// TwinCAT 3 PLC project PRG_B_Base_HMI
// Title: B_Base_HMI_Connector
// Company: RafalOS
// Author: Rafał Osajda
// ProjectVersion: 0.0.0.16
// ProgramVersion: 3.1.4026.18
// libraries:
//   B_Base, * (RafalOS)
//   Tc2_Standard, * (Beckhoff Automation GmbH)
//   Tc2_System, * (Beckhoff Automation GmbH)
//   Tc3_Module, * (Beckhoff Automation GmbH)
// project tree:
//   / PlcTask.TcTTO
//   POUs Compilation/ PRG_Compilation.TcPOU
//   POUs/A02_FB_BaseLogger_HMI/ FB_BaseLogger_HMI.TcPOU, ITF_BaseLogger_HMI.TcIO, ST_BaseLogger_HMI.TcDUT
//   POUs/A03_FB_BaseLoggerElement_HMI/ FB_BaseLoggerElement_HMI.TcPOU, ITF_BaseLoggerElement_HMI.TcIO, ST_BaseHMIConnectorEvents_ActionButtuns.TcDUT, ST_BaseHMIConnectorEvents_DetailInformation.TcDUT (not stored), ST_BaseHMIConnectorEvents_Filter.TcDUT, ST_BaseHMIConnectorEvents_ListToDisplay.TcDUT, ST_BaseLoggerElement_HMI.TcDUT, ST_BaseHMIConnectorEvents_ListToDisplayRow.TcDUT
//   POUs/A04_FB_BaseComponent_HMI/ FB_BaseComponent_HMI.TcPOU, ITF_BaseComponent_HMI.TcIO, ST_BaseComponent_HMI.TcDUT, ST_BaseComponent_HMI_Link.TcDUT
//   POUs/A05_FB_BaseControlElement_HMI/ FB_BaseControlElement_HMI.TcPOU, ITF_BaseControlElement_HMI.TcIO, ST_BaseControlElement_HMI.TcDUT, ST_BaseControlElement_HMI_Link.TcDUT
//   POUs/A06_FB_BaseGroupElement_HMI/ FB_BaseGroupElement_HMI.TcPOU, ITF_BaseGroupElement_HMI.TcIO, ST_BaseGroupElement_HMI.TcDUT, ST_BaseGroupElement_HMI_Link.TcDUT
//   POUs/A07_FB_BaseTopElement_HMI/ FB_BaseTopElement_HMI.TcPOU, ITF_BaseTopElement_HMI.TcIO, ST_BaseTopElement_HMI.TcDUT, ST_BaseTopElement_HMI_Link.TcDUT (not stored)

CONFIGURATION PRG_B_Base_HMI
    RESOURCE PLC ON TwinCAT3
        TASK PlcTask(INTERVAL := T#10ms, PRIORITY := 20);
        PROGRAM PRG_Compilation WITH PlcTask : PRG_Compilation;
    END_RESOURCE
END_CONFIGURATION

// ---- POUs/A02_FB_BaseLogger_HMI/ST_BaseLogger_HMI.TcDUT
TYPE ST_BaseLogger_HMI :
STRUCT
	bDanaBaseLogger		: BOOL;
END_STRUCT
END_TYPE

// ---- POUs/A03_FB_BaseLoggerElement_HMI/ST_BaseHMIConnectorEvents_ActionButtuns.TcDUT
(*			
	EVERDE sp. z o.o.
	Rafał Osajda		07.10.2025		TC 4024.66
	Przyciski akcji w zgłoszeniach zatwierdzanie zamykanie
*)
TYPE ST_BaseHMIConnectorEvents_ActionButtuns :
STRUCT
	bAcknowledgeAll				: BOOL;
	bAcknowledgeAllActive		: BOOL;		//widoczność przycisku 
	sAcknowledgeAll				: STRING;	//ilosci 

	bCloseAll					: BOOL;
	bCloseAllActive				: BOOL;		//widoczność przycisku 
	sCloseAll					: STRING;	//ilosci 
	
	bAcknowledgeSelected		: BOOL;
	bAcknowledgeSelectedActive	: BOOL;		//widoczność przycisku 
	sAcknowledgeSelected		: STRING;

	bCloseSelected				: BOOL;
	bCloseSelectedActive		: BOOL;		//widoczność przycisku 
	sCloseSelected				: STRING;	//ilosci 
END_STRUCT
END_TYPE

// ---- POUs/A03_FB_BaseLoggerElement_HMI/ST_BaseHMIConnectorEvents_Filter.TcDUT
TYPE ST_BaseHMIConnectorEvents_Filter :
STRUCT
	bActive						: BOOL;
	bNotActive					: BOOL;
	
	bIDItem						: BOOL;
	uiIDItem					: UINT;
	
	bIDEvent					: BOOL;
	uiIDEvent					: UINT;
	
	arrSelectedEventCategory	: ARRAY [0..GVL_BaseConstans.NUMBER_OF_EVENT_CATEGORIES] OF BOOL;	//przyciski selektora kategorii zdarzen - czy nacisniety
	arrTextOnEventCategory		: ARRAY [0..GVL_BaseConstans.NUMBER_OF_EVENT_CATEGORIES] OF STRING;	//teksty na przyciskach 
	
END_STRUCT
END_TYPE

// ---- POUs/A03_FB_BaseLoggerElement_HMI/ST_BaseHMIConnectorEvents_ListToDisplay.TcDUT
TYPE ST_BaseHMIConnectorEvents_ListToDisplay :
STRUCT
	arrToDisplay				: ARRAY [1..GVL_BaseConstans.MAX_EVENTS_TO_SHOW] OF ST_BaseHMIConnectorEvents_ListToDisplayRow;
	iNumberOfRow				: INT;
	bSelected					: BOOL;

END_STRUCT
END_TYPE

// ---- POUs/A03_FB_BaseLoggerElement_HMI/ST_BaseLoggerElement_HMI.TcDUT
TYPE ST_BaseLoggerElement_HMI :
STRUCT
	stFilter						: ST_BaseHMIConnectorEvents_Filter;
	stListOfEventsToDisplay			: ST_BaseHMIConnectorEvents_ListToDisplay;
	stButtons						: ST_BaseHMIConnectorEvents_ActionButtuns;
	stDetailInformation				: ST_BaseHMIConnectorEvents_DetailInformation;
	bSelected						: BOOL;
	iSelectedRow					: INT;
	iSelectedRowPrevius				: INT;
	bRefreshInfo					: BOOL;
	bRefreshList					: BOOL;
	
END_STRUCT
END_TYPE

// ---- POUs/A03_FB_BaseLoggerElement_HMI/ST_BaseHMIConnectorEvents_ListToDisplayRow.TcDUT
TYPE ST_BaseHMIConnectorEvents_ListToDisplayRow :
STRUCT
	uiIDEvent						: UINT;
	uiIDItem						: UINT;				//id elementu
	sCode							: STRING;			//kod elementu
	bActive							: BOOL;
	bIgnoreRepetitions				: BOOL;				//jak true nie zliczaj powtorzeń wystapienia np komunikaty
	uiRepetitionCounter				: UINT;
	sStart							: STRING;			//poczatek wystepowania zgłoszenia
	sFinish							: STRING;			//koniec wystepowaniazgloszenia
	sConfirmed						: STRING;			// stempel potwierdzenia 
	bConfirm						: BOOL;				//informacja czy potrzebne jest potwierdzenie 
	bConfirmed						: BOOL;				//pamięta czy już potwierdzone
	sEventCategory					: STRING;
	wsDescription					: WSTRING;
	wsDescriptionFull				: WSTRING;
	wsNameOfitem					: WSTRING;
END_STRUCT
END_TYPE

// ---- POUs/A04_FB_BaseComponent_HMI/ST_BaseComponent_HMI.TcDUT
TYPE ST_BaseComponent_HMI :
STRUCT
	bDanaBaseComponent		: BOOL;
	
END_STRUCT
END_TYPE

// ---- POUs/A04_FB_BaseComponent_HMI/ST_BaseComponent_HMI_Link.TcDUT
(*			
	RAFALOS
	Rafał Osajda		23.09.2025		TC 4024.66
	Struktura pomocnicza potrzeba do wiazania zmiennych
*)
TYPE ST_BaseComponent_HMI_Link :
STRUCT
	stBaseLoggerElement				: ST_BaseLoggerElement_HMI;
	stBaseComponent					: ST_BaseComponent_HMI;
END_STRUCT
END_TYPE

// ---- POUs/A05_FB_BaseControlElement_HMI/ST_BaseControlElement_HMI.TcDUT
TYPE ST_BaseControlElement_HMI :
STRUCT
	bDanaBaseControlElement		: BOOL;
	
END_STRUCT
END_TYPE

// ---- POUs/A05_FB_BaseControlElement_HMI/ST_BaseControlElement_HMI_Link.TcDUT
(*			
	RAFALOS
	Rafał Osajda		23.09.2025		TC 4024.66
	Struktura pomocnicza potrzeba do wiazania zmiennych
*)
TYPE ST_BaseControlElement_HMI_Link :
STRUCT
	stBaseLoggerElement				: ST_BaseLoggerElement_HMI;
	stBaseComponent					: ST_BaseComponent_HMI;
	stBaseControlElement			: ST_BaseControlElement_HMI;
END_STRUCT
END_TYPE

// ---- POUs/A06_FB_BaseGroupElement_HMI/ST_BaseGroupElement_HMI.TcDUT
TYPE ST_BaseGroupElement_HMI :
STRUCT
	bDanaBaseGroupElement		: BOOL;
END_STRUCT
END_TYPE

// ---- POUs/A06_FB_BaseGroupElement_HMI/ST_BaseGroupElement_HMI_Link.TcDUT
(*			
	RAFALOS
	Rafał Osajda		23.09.2025		TC 4024.66
	Struktura pomocnicza potrzeba do wiazania zmiennych
*)
TYPE ST_BaseGroupElement_HMI_Link :
STRUCT
	stBaseLoggerElement				: ST_BaseLoggerElement_HMI;
	stBaseComponent					: ST_BaseComponent_HMI;
	stBaseControlElement			: ST_BaseControlElement_HMI;
	stBaseGroupElement				: ST_BaseGroupElement_HMI;
END_STRUCT
END_TYPE

// ---- POUs/A07_FB_BaseTopElement_HMI/ST_BaseTopElement_HMI.TcDUT
TYPE ST_BaseTopElement_HMI :
STRUCT
	bDanaTopElement				: BOOL;
END_STRUCT
END_TYPE

// ---- POUs/A02_FB_BaseLogger_HMI/ITF_BaseLogger_HMI.TcIO
INTERFACE ITF_BaseLogger_HMI

END_INTERFACE

// ---- POUs/A03_FB_BaseLoggerElement_HMI/ITF_BaseLoggerElement_HMI.TcIO
INTERFACE ITF_BaseLoggerElement_HMI

(*			
	EVERDE sp. z o.o.
	Rafał Osajda		09.09.2025		TC 4024.66
	Generuje tablicę zdarzeń dla podanego ID dla 0 dla wszystkich elementów
*)
METHOD PUBLIC GetEventTableForIDItem : BOOL
VAR_INPUT
	uiIdItem			: UINT;
END_VAR
END_METHOD

(*			
	EVERDE sp. z o.o.
	Rafał Osajda		09.09.2025		TC 4024.66
	Zwraca tablicę swoich zdarzeń
*)
METHOD PUBLIC GetYourEventTable : BOOL
VAR_INPUT
END_VAR
END_METHOD

(*			
	RafalOS
	Rafał Osajda		14.11.2025		TC 4024.66
	Metoda przygotowywania danych dla HMI 
	W niej odbywa się odpytywanie właściego elementu przez łącznik
*)
METHOD PUBLIC PrepareDataForHMI : BOOL
VAR_INPUT
END_VAR
END_METHOD

END_INTERFACE

// ---- POUs/A04_FB_BaseComponent_HMI/ITF_BaseComponent_HMI.TcIO
INTERFACE ITF_BaseComponent_HMI EXTENDS ITF_BaseLogger_HMI

METHOD PUBLIC IsValidCommonData : BOOL
VAR_INPUT
END_VAR
END_METHOD

METHOD PUBLIC LinkCommonData : BOOL
VAR_INPUT
	stCommonData				: REFERENCE TO ST_BaseCommonData;
END_VAR
END_METHOD

END_INTERFACE

// ---- POUs/A05_FB_BaseControlElement_HMI/ITF_BaseControlElement_HMI.TcIO
INTERFACE ITF_BaseControlElement_HMI

END_INTERFACE

// ---- POUs/A06_FB_BaseGroupElement_HMI/ITF_BaseGroupElement_HMI.TcIO
INTERFACE ITF_BaseGroupElement_HMI EXTENDS ITF_BaseComponent_HMI

END_INTERFACE

// ---- POUs/A07_FB_BaseTopElement_HMI/ITF_BaseTopElement_HMI.TcIO
INTERFACE ITF_BaseTopElement_HMI EXTENDS ITF_BaseComponent_HMI

END_INTERFACE

// ---- POUs Compilation/PRG_Compilation.TcPOU
PROGRAM PRG_Compilation
VAR
	fbLoggerHMI				: FB_BaseLogger_HMI;
	fbLoggerElementHMI		: FB_BaseLogger_HMI;
	fbComponentHMI			: FB_BaseComponent_HMI;
	fbExecutiveElementHMI	: FB_BaseExecutiveElement_HMI;
	fbComplexElement		: FB_BaseComplexElement_HMI;
	fbMainComponent			: FB_BaseMainComponent_HMI;
END_VAR

END_PROGRAM

// ---- POUs/A02_FB_BaseLogger_HMI/FB_BaseLogger_HMI.TcPOU
(* póki co ten FB jest zbędny ale zostawiam jakby co*)
FUNCTION_BLOCK FB_BaseLogger_HMI// EXTENDS FB_Base IMPLEMENTS ITF_BaseLoggerElement_HMI
VAR
//	itfBaseLoggerConnector			: ITF_BaseLogger_HMI_Connector;	//łącznik bezpośredni do Logera
//	refstBaseLoggerDataHMI			: REFERENCE TO ST_BaseLogger_HMI;
END_VAR

END_FUNCTION_BLOCK

// ---- POUs/A04_FB_BaseComponent_HMI/FB_BaseComponent_HMI.TcPOU
FUNCTION_BLOCK FB_BaseComponent_HMI EXTENDS FB_BaseLoggerElement_HMI IMPLEMENTS ITF_BaseComponent_HMI
VAR
	itfBaseComponentConnector			: ITF_BaseComponent_HMI_Connector;
	refstBaseComponentDataHMI			: REFERENCE TO ST_BaseComponent_HMI;
END_VAR

METHOD PUBLIC IsLinkedReferences : BOOL
VAR_INPUT
END_VAR
IF (SUPER^.IsLinkedReferences () AND __ISVALIDREF (THIS^.refstBaseComponentDataHMI)) THEN
	IsLinkedReferences			:= TRUE;
END_IF
END_METHOD

END_FUNCTION_BLOCK

// ---- POUs/A03_FB_BaseLoggerElement_HMI/FB_BaseLoggerElement_HMI.TcPOU
FUNCTION_BLOCK FB_BaseLoggerElement_HMI EXTENDS FB_Base IMPLEMENTS ITF_BaseLoggerElement_HMI
VAR
	itfBaseLoggerConnector					: ITF_BaseLogger_HMI_Connector;			//bezpośredni łącznik do logera
	itfBaseLoggerElementConnector			: ITF_BaseLoggerElement_HMI_Connector;	//lacznik do FB_BaseLoggerElement np zeby wyciągnąć identyfikator
	refstBaseLoggerElementDataHMI			: REFERENCE TO ST_BaseLoggerElement_HMI;
	refstMemoryEvents						: REFERENCE TO ST_BaseEvents_Memory;	//referencja do tablicy zgłoszeń
	bIsInit									: BOOL;	//flaga informująca czy wszystkie interfejsy są dobrze przypisane
	bIsValidData							: bool;	//flaga informująca czy wszystkie dane sa podpięte 
END_VAR

METHOD PRIVATE CompleteTheDetailedInformation : BOOL
VAR_INPUT
	stRow			: ST_BaseHMIConnectorEvents_ListToDisplayRow;
END_VAR
THIS^.refstBaseLoggerElementDataHMI.stDetailInformation.uiIDEvent						:= stRow.uiIDEvent;
THIS^.refstBaseLoggerElementDataHMI.stDetailInformation.uiIDItem						:= stRow.uiIDItem;
THIS^.refstBaseLoggerElementDataHMI.stDetailInformation.sCode							:= stRow.sCode;
THIS^.refstBaseLoggerElementDataHMI.stDetailInformation.bActive							:= stRow.bActive;
THIS^.refstBaseLoggerElementDataHMI.stDetailInformation.bIgnoreRepetitions				:= stRow.bIgnoreRepetitions;
THIS^.refstBaseLoggerElementDataHMI.stDetailInformation.uiRepetitionCounter				:= stRow.uiRepetitionCounter;
THIS^.refstBaseLoggerElementDataHMI.stDetailInformation.sStart							:= stRow.sStart;
THIS^.refstBaseLoggerElementDataHMI.stDetailInformation.sFinish							:= stRow.sFinish;
THIS^.refstBaseLoggerElementDataHMI.stDetailInformation.sConfirmed						:= stRow.sConfirmed;
THIS^.refstBaseLoggerElementDataHMI.stDetailInformation.bConfirm						:= stRow.bConfirm;
THIS^.refstBaseLoggerElementDataHMI.stDetailInformation.bConfirmed						:= stRow.bConfirmed;
THIS^.refstBaseLoggerElementDataHMI.stDetailInformation.sEventCategory					:= stRow.sEventCategory;
THIS^.refstBaseLoggerElementDataHMI.stDetailInformation.wsDescription					:= stRow.wsDescription;
THIS^.refstBaseLoggerElementDataHMI.stDetailInformation.wsDescriptionFull				:= stRow.wsDescriptionFull;
END_METHOD

METHOD PRIVATE CopyDataToDisplay : BOOL
VAR_INPUT
	refarrToDisplay				: REFERENCE TO ARRAY [1..GVL_BaseConstans.MAX_EVENTS_TO_SHOW] OF ST_BaseHMIConnectorEvents_ListToDisplayRow;
	iNumberOfRow				: INT;
	stRowFromMemory				: ST_BaseEvents_RowInMemory;
	stItemInformation			: ST_BaseLogger_ItemDataToDisplay;
END_VAR
VAR
	wstmpDescriptionFull		: WSTRING;
	wstmpDescription			: WSTRING;
	iDltmp						: INT;
END_VAR
refarrToDisplay [iNumberOfRow].uiIDEvent			:= stRowFromMemory.uiIDEvent;
refarrToDisplay [iNumberOfRow].uiIDItem				:= stRowFromMemory.uiIDItem;
refarrToDisplay [iNumberOfRow].bActive				:= stRowFromMemory.bActive;
refarrToDisplay [iNumberOfRow].sCode				:= stItemInformation.sCode; 
refarrToDisplay [iNumberOfRow].bIgnoreRepetitions	:= stRowFromMemory.bIgnoreRepetitions;
refarrToDisplay [iNumberOfRow].bConfirm				:= stRowFromMemory.bConfirm;
refarrToDisplay [iNumberOfRow].bConfirmed			:= stRowFromMemory.bConfirmed;

refarrToDisplay [iNumberOfRow].sStart				:= THIS^.refstCommonData.itfTime.BaseDTToString (inDT := stRowFromMemory.dtStart);
IF (TO_STRING (stRowFromMemory.dtConfirmed) <> 'DT#1970-01-01-00:00:00') THEN
	refarrToDisplay [iNumberOfRow].sConfirmed		:= THIS^.refstCommonData.itfTime.BaseDTToString (inDT := stRowFromMemory.dtConfirmed);
ELSE
	refarrToDisplay [iNumberOfRow].sConfirmed		:= '';
END_IF
IF (TO_STRING (TO_STRING (stRowFromMemory.dtFinish)) <> 'DT#1970-01-01-00:00:00') THEN
	refarrToDisplay [iNumberOfRow].sFinish			:= THIS^.refstCommonData.itfTime.BaseDTToString (inDT := stRowFromMemory.dtFinish);
ELSE
	refarrToDisplay [iNumberOfRow].sFinish			:= '';
END_IF

refarrToDisplay [iNumberOfRow].sEventCategory		:= stItemInformation.sEventCategory; 
refarrToDisplay [iNumberOfRow].uiRepetitionCounter	:= stItemInformation.uiRepetitionCounter;
wstmpDescriptionFull		:= THIS^.GetTextFromLabelForActiveLocation (stLabel	:= stItemInformation.stDescription);
iDltmp												:= WLEN (wstmpDescriptionFull);
IF (iDltmp > 100) THEN
	wstmpDescription								:= WDELETE (wstmpDescriptionFull, iDltmp - 100, iDltmp);
END_IF
refarrToDisplay [iNumberOfRow].wsDescription		:= wstmpDescription;
refarrToDisplay [iNumberOfRow].wsDescriptionFull	:= wstmpDescriptionFull;
refarrToDisplay [iNumberOfRow].wsNameOfitem			:= THIS^.GetTextFromLabelForActiveLocation (stLabel := stItemInformation.stItemName);
END_METHOD

METHOD PUBLIC CreateLinkToEventsMemory : BOOL
VAR_INPUT
END_VAR
THIS^.refstMemoryEvents	REF= THIS^.itfBaseLoggerConnector.GetReferenceToStmemory ();


IF (__ISVALIDREF (THIS^.refstMemoryEvents)) THEN
	CreateLinkToEventsMemory		:= TRUE;
ELSE
	CreateLinkToEventsMemory		:= FALSE;
END_IF
END_METHOD

(*			
	EVERDE sp. z o.o.
	Rafał Osajda		09.09.2025		TC 4024.66
	Generuje tablicę zdarzeń dla podanego ID dla 0 dla wszystkich elementów
*)
METHOD PUBLIC GetEventTableForIDItem : BOOL
VAR_INPUT
	uiIdItem				: UINT;
END_VAR
VAR_INST
	bFilterIsActivePrevius	: BOOL;	
END_VAR
VAR
	iI						: INT;
	bFilterIsActive			: BOOL;
	bUsunZListy				: BOOL;
	btmpUsunZListy			: BOOL;
	refstMemory				: REFERENCE TO ST_BaseEvents_Memory;
	refstListToDisplay		: REFERENCE TO ST_BaseHMIConnectorEvents_ListToDisplay;
	refstFilter				: REFERENCE TO ST_BaseHMIConnectorEvents_Filter;
	refstActionButtons		: REFERENCE TO ST_BaseHMIConnectorEvents_ActionButtuns;
	stRowFromMemory			: ST_BaseEvents_RowInMemory;
	stItemInformation		: ST_BaseLogger_ItemDataToDisplay;
(*	Ilosci zdarzen wyswietlanych na liscie	*)
	stNumberEventToDisplay	: ST_BaseEvents_ActiveEvents;
//
	iIAck: INT;
	iIClose: INT;
END_VAR
(*
	sprawdzenie czy jest coś nowego - tak generuj
	jak już jest wygenerowana jakaś lista i zmienił się filtr - tak to generuj

*)
IF (THIS^.refstMemoryEvents.iNumberOfRow > 0) THEN

	refstMemory				REF= THIS^.refstMemoryEvents;
	refstListToDisplay		REF= THIS^.refstBaseLoggerElementDataHMI.stListOfEventsToDisplay;
	refstFilter				REF= THIS^.refstBaseLoggerElementDataHMI.stFilter;
	refstActionButtons		REF= THIS^.refstBaseLoggerElementDataHMI.stButtons;
	bFilterIsActive			:= GetIsActiveFilter (refstFilter := refstFilter);		//sprawdzenie czy jest aktywny filtr
	
	IF (THIS^.itfBaseLoggerConnector.GetChangeInMemory () OR bFilterIsActive 
		OR bFilterIsActivePrevius OR THIS^.refstBaseLoggerElementDataHMI.bRefreshList) THEN
		THIS^.refstBaseLoggerElementDataHMI.bRefreshList	:= FALSE;
		bFilterIsActivePrevius								:= bFilterIsActive;

		THIS^.itfBaseLoggerConnector.ResetChangeInMemory ();
		(*	Wyczyszczenie tablicy wyświetlania		*)
		Tc2_System.MEMSET (
			destAddr		:= ADR (refstListToDisplay.arrToDisplay),
			fillByte		:= 0,
			n				:= SIZEOF (refstListToDisplay.arrToDisplay)
		);
		refstListToDisplay.iNumberOfRow		:= 0;
		FOR iI := 1 TO refstMemory.iNumberOfRow DO
			IF (uiIdItem = refstMemory.arrRow [iI].uiIDItem OR uiIdItem = 0) THEN
				stRowFromMemory			:= refstMemory.arrRow [iI];
				stItemInformation		:= THIS^.itfBaseLoggerConnector.GetInformationFromItem (uiIDItem := uiIdItem, uiIDEvent := stRowFromMemory.uiIDEvent);
				bUsunZListy		:= THIS^.RemoveRowFormList (
										refstFilter 		:= refstFilter, 
										uiIDEvent 			:= stRowFromMemory.uiIDEvent, 
										uiIDItem 			:=  stRowFromMemory.uiIDItem,
										bActive				:= stRowFromMemory.bActive,
										stItemInformation	:= stItemInformation
									);
				IF (NOT bUsunZListy) THEN
					refstListToDisplay.iNumberOfRow		:= refstListToDisplay.iNumberOfRow + 1;
					THIS^.CopyDataToDisplay (
						refarrToDisplay					:= refstListToDisplay.arrToDisplay,
						iNumberOfRow					:= refstListToDisplay.iNumberOfRow,
						stRowFromMemory					:= stRowFromMemory,
						stItemInformation				:= stItemInformation
					);
	(*	Informacja o ilosciach zgloszen na wyswietlanej liście 		*)
					stNumberEventToDisplay.iTotalNumer	:= stNumberEventToDisplay.iTotalNumer + 1;
					IF (refstListToDisplay.arrToDisplay [refstListToDisplay.iNumberOfRow].bActive) THEN
						stNumberEventToDisplay.iNumberOfActive	:= stNumberEventToDisplay.iNumberOfActive + 1;
						stNumberEventToDisplay.arrNumberOfActive [stItemInformation.eEventCategory] := stNumberEventToDisplay.arrNumberOfActive [stItemInformation.eEventCategory] + 1;
						stNumberEventToDisplay.arrActive [stItemInformation.eEventCategory]	:= TRUE;
					END_IF
					IF (refstListToDisplay.arrToDisplay [refstListToDisplay.iNumberOfRow].bConfirm AND 
						NOT refstListToDisplay.arrToDisplay [refstListToDisplay.iNumberOfRow].bConfirmed) THEN
						stNumberEventToDisplay.iNumberOfActiveWithConfirmation	:= stNumberEventToDisplay.iNumberOfActiveWithConfirmation + 1;
					END_IF
					stNumberEventToDisplay.arrTotalNumer [stItemInformation.eEventCategory] := stNumberEventToDisplay.arrTotalNumer [stItemInformation.eEventCategory] + 1;
				END_IF	//usuwanie z listy
			END_IF
	(*	Liczba zgłoszeń większa od tych co wyświetlamy	starsze można zobaczyć na kompie po podłaczeniu 	*)
			IF (refstListToDisplay.iNumberOfRow = TO_INT (GVL_BaseConstans.MAX_EVENTS_TO_SHOW)) THEN
				EXIT;
			END_IF
		END_FOR	//koniec przechodzenia przez wiersze pamięci
	(*	Informacja o ilosciach zgloszen		*)
		IF (uiIdItem > 0) THEN
			THIS^.PrepareQuantitiesForDisplay (
				stCounted		:= stNumberEventToDisplay,
				stFromLogger	:= THIS^.itfBaseLoggerConnector.GetEventCountsForItem (uiIDItem := uiIDItem)
			);
		ELSE
			THIS^.PrepareQuantitiesForDisplay (
				stCounted		:= stNumberEventToDisplay,
				stFromLogger	:= THIS^.itfBaseLoggerConnector.GetEventCounts ()
			);
		END_IF
		refstActionButtons.bAcknowledgeAllActive	:= stNumberEventToDisplay.iNumberOfActiveWithConfirmation > 0;
		refstActionButtons.bCloseAllActive			:= stNumberEventToDisplay.iNumberOfActive > 0;
	END_IF
	IF (THIS^.refstBaseLoggerElementDataHMI.bSelected) THEN
		refstActionButtons.bAcknowledgeSelectedActive	:= refstListToDisplay.arrToDisplay [THIS^.refstBaseLoggerElementDataHMI.iSelectedRow].bConfirm AND 
			NOT refstListToDisplay.arrToDisplay [THIS^.refstBaseLoggerElementDataHMI.iSelectedRow].bConfirmed;
		refstActionButtons.bCloseSelectedActive			:= refstListToDisplay.arrToDisplay [THIS^.refstBaseLoggerElementDataHMI.iSelectedRow].bConfirm AND 
			refstListToDisplay.arrToDisplay [THIS^.refstBaseLoggerElementDataHMI.iSelectedRow].bConfirmed;
	ELSE
		refstActionButtons.bAcknowledgeSelectedActive	:= FALSE;
		refstActionButtons.bCloseSelectedActive			:= FALSE;
	END_IF
	
	(*	Wybor zgloszenia z listy	*)

	IF ((THIS^.refstBaseLoggerElementDataHMI.iSelectedRow <> THIS^.refstBaseLoggerElementDataHMI.iSelectedRowPrevius AND
		THIS^.refstBaseLoggerElementDataHMI.bSelected) OR THIS^.refstBaseLoggerElementDataHMI.bRefreshInfo ) THEN
		THIS^.CompleteTheDetailedInformation (stRow := refstListToDisplay.arrToDisplay [THIS^.refstBaseLoggerElementDataHMI.iSelectedRow]);
	ELSIF (NOT THIS^.refstBaseLoggerElementDataHMI.bSelected) THEN
		THIS^.refstBaseLoggerElementDataHMI.iSelectedRow		:= -1;
		THIS^.refstBaseLoggerElementDataHMI.iSelectedRowPrevius	:= -1;
	END_IF 
	
	(*	Obsługa przycisków zamykania i potwierrdzania zgłoszeń	*)

	IF (THIS^.refstBaseLoggerElementDataHMI.stButtons.bAcknowledgeSelected) THEN //potwierdz zgłoszenie
		IF (refstListToDisplay.arrToDisplay [THIS^.refstBaseLoggerElementDataHMI.iSelectedRow].bConfirm AND 
			NOT refstListToDisplay.arrToDisplay [THIS^.refstBaseLoggerElementDataHMI.iSelectedRow].bConfirmed) THEN
			THIS^.itfBaseLoggerElementConnector.EventAcknowledgeByID (uiIDEvent := THIS^.refstBaseLoggerElementDataHMI.stDetailInformation.uiIDEvent);
		END_IF
	END_IF

	IF (THIS^.refstBaseLoggerElementDataHMI.stButtons.bCloseSelected) THEN	//zamknij zgłoszenie
		IF (refstListToDisplay.arrToDisplay [THIS^.refstBaseLoggerElementDataHMI.iSelectedRow].bActive OR 
			refstListToDisplay.arrToDisplay [THIS^.refstBaseLoggerElementDataHMI.iSelectedRow].sFinish <> '') THEN
			THIS^.itfBaseLoggerElementConnector.EventSetInactiveByID (uiIDEvent := THIS^.refstBaseLoggerElementDataHMI.stDetailInformation.uiIDEvent);
		END_IF
	END_IF

	IF (THIS^.refstBaseLoggerElementDataHMI.stButtons.bAcknowledgeAll) THEN //potwierdz wszystkie niepotwierdzone zgłoszenie
		FOR iIAck := 1 TO TO_INT (refstListToDisplay.iNumberOfRow) DO
			IF (refstListToDisplay.arrToDisplay [iIAck].bConfirm AND 
				NOT refstListToDisplay.arrToDisplay [iIAck].bConfirmed) THEN
				THIS^.itfBaseLoggerElementConnector.EventAcknowledgeByID (uiIDEvent := refstListToDisplay.arrToDisplay [iIAck].uiIDEvent);
			END_IF
		END_FOR
	END_IF
	IF (THIS^.refstBaseLoggerElementDataHMI.stButtons.bCloseAll) THEN	//zamknij wszystkie nie zamnknięte zgłoszenie
		FOR iIClose := 1 TO TO_INT (refstListToDisplay.iNumberOfRow) DO
			IF (refstListToDisplay.arrToDisplay [iIClose].bActive OR refstListToDisplay.arrToDisplay [iIClose].sFinish <> '') THEN
				THIS^.itfBaseLoggerElementConnector.EventSetInactiveByID (uiIDEvent := refstListToDisplay.arrToDisplay [iIClose].uiIDEvent);
			END_IF
		END_FOR
	END_IF
	
	
	THIS^.refstBaseLoggerElementDataHMI.bRefreshList		:= 	refstActionButtons.bAcknowledgeSelected OR
																refstActionButtons.bCloseSelected OR
																refstActionButtons.bAcknowledgeAll OR
																refstActionButtons.bCloseAll;
	THIS^.refstBaseLoggerElementDataHMI.bRefreshInfo		:= 	refstActionButtons.bAcknowledgeSelected	OR
																refstActionButtons.bCloseSelected OR
	                                                          	refstActionButtons.bAcknowledgeAll OR
                                                               	refstActionButtons.bCloseAll;
	refstActionButtons.bAcknowledgeSelected					:= FALSE;
	refstActionButtons.bCloseSelected						:= FALSE;
	refstActionButtons.bAcknowledgeAll						:= FALSE;
	refstActionButtons.bCloseAll							:= FALSE;

END_IF
END_METHOD

METHOD PRIVATE GetIsActiveFilter : BOOL
VAR_INPUT
	refstFilter				: REFERENCE TO ST_BaseHMIConnectorEvents_Filter;
END_VAR
VAR
	bResult: BOOL;
	iI: INT;
END_VAR
bResult				:= refstFilter.bActive OR 
						refstFilter.bNotActive OR
						refstFilter.bIDEvent OR
						refstFilter.bIDItem;
FOR iI := 1 TO GVL_BaseConstans.NUMBER_OF_EVENT_CATEGORIES DO
	bResult			:= bResult OR refstFilter.arrSelectedEventCategory [iI];
END_FOR

GetIsActiveFilter	:= bResult;
END_METHOD

METHOD PROTECTED GetTextFromLabel : WSTRING
VAR_INPUT
	stLabel				: ST_BaseLabel;
	eLocation			: E_BaseLocation;
END_VAR
GetTextFromLabel := stLabel.arrText [eLocation];
END_METHOD

METHOD PROTECTED GetTextFromLabelForActiveLocation : WSTRING
VAR_INPUT
	stLabel				: ST_BaseLabel;
END_VAR

VAR
	dfsfsdaf: WSTRING;
END_VAR
GetTextFromLabelForActiveLocation := stLabel.arrText [THIS^.refstCommonData.itfLocaciotn.GetLocation ()];
END_METHOD

(*			
	EVERDE sp. z o.o.
	Rafał Osajda		09.09.2025		TC 4024.66
	Zwraca tablicę swoich zdarzeń
*)
METHOD PUBLIC GetYourEventTable : BOOL
VAR_INPUT
END_VAR
THIS^.GetEventTableForIDItem (uiIdItem := THIS^.itfBaseLoggerElementConnector.GetID ());		//przygotowanie tablicy dla siebie
END_METHOD

(*			
	RAFALOS
	Rafał Osajda		23.09.2025		TC 4024.66
	Zwraca informację czy dane są podpięte do systemu
*)
METHOD PUBLIC IsInit : BOOL
VAR_INPUT
END_VAR
IsInit			:= THIS^.bIsInit;
END_METHOD

METHOD PUBLIC IsLinkedReferences : BOOL
VAR_INPUT
END_VAR
IF (__ISVALIDREF (THIS^.refstBaseLoggerElementDataHMI)) THEN
	IsLinkedReferences			:= TRUE;
END_IF
END_METHOD

(*			
	RAFALOS
	Rafał Osajda		23.09.2025		TC 4024.66
	Zwraca flagę przypisywaną w FB_Init tworzonego elementu
*)
METHOD IsValidData : BOOL
VAR_INPUT
END_VAR
IsValidData				:= THIS^.bIsValidData;
END_METHOD

(*			
	RafalOS
	Rafał Osajda		14.11.2025		TC 4024.66
	Metoda przygotowywania danych dla HMI 
	W niej odbywa się odpytywanie właściego elementu przez łącznik
*)
METHOD PUBLIC PrepareDataForHMI : BOOL
VAR_INPUT
END_VAR
END_METHOD

METHOD PRIVATE PrepareQuantitiesForDisplay : BOOL
VAR_INPUT
	stCounted			: ST_BaseEvents_ActiveEvents;
	stFromLogger		: ST_BaseEvents_ActiveEvents;
END_VAR

VAR
	iI: INT;
	stmp1: STRING;
END_VAR
stmp1	:= CONCAT (stmp1,TO_STRING (stCounted.iNumberOfActiveWithConfirmation));
stmp1	:= CONCAT (stmp1, '/');
stmp1	:= CONCAT (stmp1, TO_STRING (stFromLogger.iNumberOfActiveWithConfirmation));

THIS^.refstBaseLoggerElementDataHMI.stButtons.sAcknowledgeAll		:= stmp1;
THIS^.refstBaseLoggerElementDataHMI.stButtons.sAcknowledgeSelected	:= '1/1';

stmp1	:= CONCAT ('',TO_STRING (stCounted.iNumberOfActive));
stmp1	:= CONCAT (stmp1, '/');
stmp1	:= CONCAT (stmp1, TO_STRING (stFromLogger.iNumberOfActive));
THIS^.refstBaseLoggerElementDataHMI.stButtons.sCloseAll				:= stmp1;
THIS^.refstBaseLoggerElementDataHMI.stButtons.sCloseSelected		:= '1/1';

FOR iI := 1	TO GVL_BaseConstans.NUMBER_OF_EVENT_CATEGORIES DO
	THIS^.refstBaseLoggerElementDataHMI.stFilter.arrTextOnEventCategory [iI]	:= 
		CONCAT (TO_STRING (stCounted.arrTotalNumer [iI]), CONCAT ('/',TO_STRING (stFromLogger.arrTotalNumer [iI])));
END_FOR
END_METHOD

METHOD PRIVATE RemoveRowFormList : BOOL
VAR_INPUT
	refstFilter				: REFERENCE TO ST_BaseHMIConnectorEvents_Filter;
	uiIDEvent				: UINT;
	uiIDItem				: UINT;
	bActive					: BOOL;
	stItemInformation		: ST_BaseLogger_ItemDataToDisplay;
END_VAR
VAR
	bRemove					: BOOL;
	iK						: INT;
	bRemoveHelp				: BOOL;
END_VAR
bRemove		:= FALSE;
bRemove		:= bRemove OR (refstFilter.bActive AND NOT bActive);
bRemove		:= bRemove OR (refstFilter.bNotActive AND bActive);
bRemove		:= bRemove OR (refstFilter.bIDItem	AND uiIDItem <> refstFilter.uiIDItem);
bRemove		:= bRemove OR (refstFilter.bIDEvent AND 
uiIDEvent <> refstFilter.uiIDEvent);
FOR iK := 1 TO GVL_BaseConstans.NUMBER_OF_EVENT_CATEGORIES DO
	CASE iK OF 
		E_BaseEvents_Category.Error		: bRemoveHelp	:=  stItemInformation.eEventCategory = E_BaseEvents_Category.Error;
		E_BaseEvents_Category.Alarm		: bRemoveHelp	:=  stItemInformation.eEventCategory = E_BaseEvents_Category.Alarm;
		E_BaseEvents_Category.Safety	: bRemoveHelp	:=  stItemInformation.eEventCategory = E_BaseEvents_Category.Safety;
		E_BaseEvents_Category.Message	: bRemoveHelp	:=  stItemInformation.eEventCategory = E_BaseEvents_Category.Message;
	END_CASE
	bRemove		:= bRemove OR (refstFilter.arrSelectedEventCategory [iK] AND bRemoveHelp);
END_FOR
//przeddział czasowy

RemoveRowFormList	:= bRemove;
END_METHOD

METHOD PROTECTED SelectLocation : WSTRING
VAR_INPUT
	stTexts			: ST_BaseLabel;
	eLocation		: E_BaseLocation;
END_VAR
SelectLocation := stTexts.arrText [eLocation];
END_METHOD

END_FUNCTION_BLOCK

// ---- POUs/A05_FB_BaseControlElement_HMI/FB_BaseControlElement_HMI.TcPOU
FUNCTION_BLOCK FB_BaseControlElement_HMI EXTENDS FB_BaseComponent_HMI IMPLEMENTS ITF_BaseControlElement_HMI
VAR
	itfBaseControlElementConnector		: ITF_BaseControlElement_HMI_Connector;
	refstBaseControlElementDataHMI		: REFERENCE TO ST_BaseControlElement_HMI;
	(*	lista componentów składających się na ten element w elemencie docelowym dodać itf dla konkretnych elementów	*)
	arrComponent						: ARRAY  [1..GVL_BaseConstans.MAX_ITEM_PER_ELEMENT] OF ITF_BaseComponent_HMI;
	uiNumberOfComponents				: UINT;

END_VAR

METHOD PROTECTED AddComponent : BOOL
VAR_INPUT
	itfComponentHMI				: ITF_BaseComponent_HMI;
END_VAR
IF (THIS^.uiNumberOfComponents + 1 <= GVL_BaseConstans.MAX_ITEM_PER_ELEMENT) THEN
	THIS^.uiNumberOfComponents		:= THIS^.uiNumberOfComponents + 1;
	THIS^.arrComponent [THIS^.uiNumberOfComponents]	:= itfComponentHMI;
	AddComponent				:= TRUE;
ELSE
	;//zwrocenie zbyt dużo komponentow
END_IF
END_METHOD

END_FUNCTION_BLOCK

// ---- POUs/A06_FB_BaseGroupElement_HMI/FB_BaseGroupElement_HMI.TcPOU
FUNCTION_BLOCK FB_BaseGroupElement_HMI EXTENDS FB_BaseControlElement_HMI IMPLEMENTS ITF_BaseGroupElement_HMI
VAR
	itfBaseGroupElementConnector		: ITF_BaseGroupElement_HMI_Connector;
	refstBaseGroupElementDataHMI		: REFERENCE TO ST_BaseGroupElement_HMI;
	(*	lista elementów składających się na ten element w elemencie docelowym dodać itf dla konkretnych elementów	*)
	arrControlElement					: ARRAY [1..GVL_BaseConstans.MAX_ITEM_PER_ELEMENT] OF ITF_BaseControlElement_HMI;
	uiNumberOfControlElement			: UINT;
END_VAR

METHOD PROTECTED AddControlElement : BOOL
VAR_INPUT
	itfControlElementHMI		: ITF_BaseControlElement_HMI;
END_VAR
IF (THIS^.uiNumberOfControlElement + 1 <= GVL_BaseConstans.MAX_ITEM_PER_ELEMENT) THEN
	THIS^.uiNumberOfControlElement		:= THIS^.uiNumberOfControlElement + 1;
	THIS^.arrControlElement [THIS^.uiNumberOfControlElement]	:= itfControlElementHMI;
	AddControlElement			:= TRUE;
ELSE
	;//zwrocenie zbyt dużo komponentow
END_IF
END_METHOD

METHOD PUBLIC IsLinkedReferences : BOOL
VAR_INPUT
END_VAR
IF (SUPER^.IsLinkedReferences () AND __ISVALIDREF (THIS^.refstBaseGroupElementDataHMI)) THEN
	IsLinkedReferences			:= TRUE;
END_IF
END_METHOD

METHOD PUBLIC IsValidCommonData : BOOL
VAR_INPUT
END_VAR

VAR
	bResult: BOOL;
	iI: INT;
END_VAR
bResult						:= SUPER^.IsValidCommonData ();

FOR iI := 1 TO TO_INT (THIS^.uiNumberOfControlElement) DO
	bResult					:= bResult AND THIS^.arrControlElement [iI].IsValidCommonData ();
END_FOR

IsValidCommonData			:= bResult;
END_METHOD

METHOD PUBLIC LinkCommonData : BOOL
VAR_INPUT
	stCommonData				: REFERENCE TO ST_BaseCommonData;
END_VAR
VAR
	bResult						: BOOL;
	iI: INT;
END_VAR
bResult							:= SUPER^.LinkCommonData (stCommonData := stCommonData);

FOR iI := 1 TO TO_INT (THIS^.uiNumberOfControlElement) DO
	bResult := bResult AND THIS^.arrControlElement [iI].LinkCommonData (stCommonData := stCommonData);
END_FOR

LinkCommonData					:= bResult;
END_METHOD

END_FUNCTION_BLOCK

// ---- POUs/A07_FB_BaseTopElement_HMI/FB_BaseTopElement_HMI.TcPOU
FUNCTION_BLOCK FB_BaseTopElement_HMI EXTENDS FB_BaseGroupElement_HMI IMPLEMENTS ITF_BaseTopElement_HMI
VAR
	itfBaseTopElementConnector			: ITF_BaseTopElement_HMI_Connector;
	refstBaseTopElementDataHMI			: REFERENCE TO ST_BaseTopElement_HMI;
END_VAR

METHOD PUBLIC IsLinkedReferences : BOOL
VAR_INPUT
END_VAR
IF (SUPER^.IsLinkedReferences () AND __ISVALIDREF (THIS^.refstBaseTopElementDataHMI)) THEN
	IsLinkedReferences			:= TRUE;
END_IF
END_METHOD

END_FUNCTION_BLOCK
